FUNCTION_BLOCK UA_WriteWrapper IMPLEMENTS I_OPCUA_Write
VAR_INPUT
END_VAR
VAR_OUTPUT
END_VAR
VAR
	uaWrite : UA_Write;
END_VAR

{warning 'add method implementation '}
METHOD start : BOOL
VAR_INPUT
	Execute	: BOOL;
	ConnectionHdl	: DWORD;
	NodeHdl	: DWORD;
	stNodeAddInfo	: Tc3_PLCopen_OpcUa.ST_UANodeAdditionalInfo;
	pVariable	: PVOID;
	cbData	: UDINT;
	Timeout	: TIME := DEFAULT_ADS_TIMEOUT;
END_VAR
VAR_OUTPUT
	Done	: BOOL;
	Busy	: BOOL;
	Error	: BOOL;
	ErrorID	: DWORD;
END_VAR
uaWrite(Execute := execute,
		 COnnectionhdl := connectionhdl, 
		NodeHdl := nodehdl, 
		stNodeAddInfo := stnodeaddinfo, 
		pVariable := pvariable, 
		cbdata := cbData, 
		Timeout := timeout,
		Done => DOne,
		Busy => Busy,
		Error => Error,
		ErrorID => ErrorID
		);
END_METHOD

END_FUNCTION_BLOCK

(* stored: Version 1.1.0.1, ProductVersion 3.1.4024.9
   POU UA_WriteWrapper: Id {c5574620-7228-43d8-a779-cd023918d3b1}, SpecialFunc None
   Method start: Id {e36f055a-29cb-4751-a4e9-8075ddd205ec} *)
